INTERFACE I_CalcXRayDelta EXTENDS I_Fallible


METHOD Calculate
VAR_INPUT
    MaterialFormula : T_MaxString;
    Delta : I_QuantityLREALPublic;
END_VAR
END_METHOD

END_INTERFACE

(* stored: Version 1.1.0.1
   Itf I_CalcXRayDelta: Id {dc69db79-eeb2-42dd-978a-33fdd2556306}
   Method Calculate: Id {d40de753-cc51-40d1-ae5d-ee3d341a0999} *)
